METHOD metNotShowChannel : BOOL
VAR_INPUT
    iChannel    :   INT;
END_VAR
IF iChannel >= 1 AND iChannel <= 16 THEN
    metNotShowChannel := NOT ayShowChanel[iChannel];
ELSE
    metNotShowChannel := TRUE;
END_IF
END_METHOD

PROPERTY proScrollBar : INT
SET
iScrollBar := proScrollBar;
END_SET
GET
proScrollBar := iOldScrollBar;
END_GET
END_PROPERTY

METHOD PRIVATE metCalcScrollBar : INT
VAR_INPUT
    usiSlot :   USINT;
END_VAR
IF usiSlot <= 11 THEN
    metCalcScrollBar := 0;
ELSE
    metCalcScrollBar := TO_INT(LIMIT(0,((usiSlot -11)* TO_INT(rFactor * 49)),TO_INT(rFactor *2921)));
END_IF;
END_METHOD

METHOD PRIVATE metCalcSlotFromScrollBar : USINT
VAR_INPUT
    iScrollBarIn  :   INT;
END_VAR
IF iScrollBarIn / 49 <= 11 THEN
    metCalcSlotFromScrollBar := 11;
ELSE
    metCalcSlotFromScrollBar := TO_USINT(iScrollBarIn / MAX(1,TO_INT(rFactor*49)));
END_IF;
END_METHOD

METHOD getSizeOfFrame : BOOL
VAR_INPUT
	ptIn	:	VisuElems.VisuStructPoint;
END_VAR
getSizeOfFrame := FALSE;
iFrameSize := ptIn.iX;

IF iFrameSize > 0 THEN
	rFactor := TO_REAL(iFrameSize) / 3000.0;
ELSE
	rFactor := 0;
END_IF
END_METHOD

END_FUNCTION_BLOCK

// 40 Visualizations/AI/SimAI_Temp
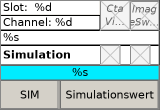
VISUALIZATION SimAI_Temp  // 160x110
VAR_INPUT
	ITF_AI : ITF_AI;
END_VAR
VAR_IN_OUT
	IO_Ref_In	:	fbAI;
END_VAR
    Frame (0,0 160x45)
        shows ModulInfos(ITF_IO := ITF_AI)
    Frame (0,45 160x20)
        shows SimulationInfos(ITF_IO_REF_IN := ITF_AI.proThisRef_AI)
    Textfield (0,65 160x15), "%s", text variable: ITF_AI.proPhysikalValueVisu
    Button (0,80 60x30), "SIM", colour toggle: IO_Ref_In.fbxSimulation.xValue, pressed state: IO_Ref_In.fbxSimulation.xValue, invisible if: IO_Ref_In.fbxSimulationLock.xValue
        toggle IO_Ref_In.fbxSimulation.xValue
    Button (60,80 100x30), "Simulationswert", text variable: IO_Ref_In.fbrSimulationValue.rValue, invisible if: IO_Ref_In.fbxSimulationLock.xValue OR NOT IO_Ref_In.fbxSimulation.xValue
        OnMouseClick: write the text variable via InputWithLimits, min GlobalKonstant.ayMin[ITF_AI.proModuleType], max GlobalKonstant.ayMax[ITF_AI.proModuleType]
END_VISUALIZATION

// 40 Visualizations/AI/SimAI
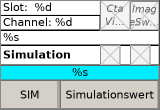
VISUALIZATION SimAI  // 160x110
VAR_INPUT	
	ITF_AI : ITF_AI;
END_VAR
    Frame (0,0 160x110), invisible if: NOT __QUERYINTERFACE(ITF_AI,ITF_AI)
        shows SimAI_Temp_Querry(ITF_AI := ITF_AI)
END_VISUALIZATION

// 40 Visualizations/AO/SimAO_Temp
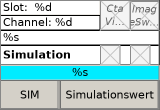
VISUALIZATION SimAO_Temp  // 160x110
VAR_INPUT
	ITF_AO : ITF_AO;
END_VAR
VAR_IN_OUT
	IO_Ref_In	:	fbAO;
END_VAR
    Frame (0,0 160x45)
        shows ModulInfos(ITF_IO := ITF_AO)
    Frame (0,45 160x20)
        shows SimulationInfos(ITF_IO_REF_IN := ITF_AO.proThisRef_AO)
    Textfield (0,65 160x15), "%s", text variable: ITF_AO.proPhysikalValueVisu
    Button (0,80 60x30), "SIM", colour toggle: IO_Ref_In.fbxSimulation.xValue, pressed state: IO_Ref_In.fbxSimulation.xValue, invisible if: IO_Ref_In.fbxSimulationLock.xValue
        toggle IO_Ref_In.fbxSimulation.xValue
    Button (60,80 100x30), "Simulationswert", text variable: IO_Ref_In.fbrSimulationValue.rValue, invisible if: IO_Ref_In.fbxSimulationLock.xValue OR NOT IO_Ref_In.fbxSimulation.xValue
        OnMouseClick: write the text variable via InputWithLimits, min GlobalKonstant.ayMin[ITF_AO.proModuleType], max GlobalKonstant.ayMax[ITF_AO.proModuleType]
END_VISUALIZATION

// 40 Visualizations/AO/SimAO
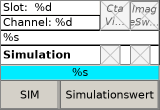
VISUALIZATION SimAO  // 160x110
VAR_INPUT	
	ITF_AO : ITF_AO;
END_VAR
    Frame (0,0 160x110), invisible if: NOT __QUERYINTERFACE(ITF_AO,ITF_AO)
        shows SimAO_Temp_Querry(ITF_AO := ITF_AO)
END_VISUALIZATION

// 40 Visualizations/DI/SimDI
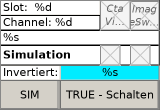
VISUALIZATION SimDI  // 160x110
VAR_INPUT	
	ITF_DI : ITF_DI;
END_VAR
    Frame (0,0 160x110), invisible if: NOT __QUERYINTERFACE(ITF_DI,ITF_DI)
        shows SimDI_Temp_Querry(ITF_DI := ITF_DI)
END_VISUALIZATION

// 40 Visualizations/DI/SimDI_Temp
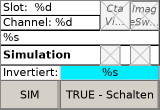
VISUALIZATION SimDI_Temp  // 160x110
VAR_INPUT
	ITF_DI : ITF_DI;
END_VAR
VAR_IN_OUT
	IO_Ref_In	:	fbDI;
END_VAR
    Textfield (0,65 60x15), colour toggle: IO_Ref_In.fbxInvert.xValue
    Textfield (60,65 100x15), "%s", text variable: ITF_DI.proPhysikalValueVisu
    Label (0,65 60x15), "Invertiert:", invisible if: NOT IO_Ref_In.fbxInvert.xValue
    Button (0,80 60x30), "SIM", colour toggle: IO_Ref_In.fbxSimulation.xValue, pressed state: IO_Ref_In.fbxSimulation.xValue, invisible if: IO_Ref_In.fbxSimulationLock.xValue
        toggle IO_Ref_In.fbxSimulation.xValue
    Button (60,80 100x30), "FALSE - Schalten", pressed state: IO_Ref_In.fbxSimulationValue.xValue, invisible if: IO_Ref_In.fbxSimulationLock.xValue OR NOT IO_Ref_In.fbxSimulation.xValue OR NOT IO_Ref_In.fbxSimulationValue.xValue OR IO_Ref_In.fbxInvert.xValue
        toggle IO_Ref_In.fbxSimulationValue.xValue p2164770859=TRUE
    Frame (0,0 160x45)
        shows ModulInfos(ITF_IO := ITF_DI)
    Frame (0,45 160x20)
        shows SimulationInfos(ITF_IO_REF_IN := ITF_DI.proThisRef_DI)
    Button (60,80 100x30), "TRUE - Schalten", pressed state: IO_Ref_In.fbxSimulationValue.xValue, invisible if: IO_Ref_In.fbxSimulationLock.xValue OR NOT IO_Ref_In.fbxSimulation.xValue OR IO_Ref_In.fbxSimulationValue.xValue OR IO_Ref_In.fbxInvert.xValue
        toggle IO_Ref_In.fbxSimulationValue.xValue
    Button (60,80 100x30), "FALSE - Schalten", pressed state: IO_Ref_In.fbxSimulationValue.xValue, invisible if: IO_Ref_In.fbxSimulationLock.xValue OR NOT IO_Ref_In.fbxSimulation.xValue OR IO_Ref_In.fbxSimulationValue.xValue OR NOT IO_Ref_In.fbxInvert.xValue
        toggle IO_Ref_In.fbxSimulationValue.xValue
    Button (60,80 100x30), "TRUE - Schalten", pressed state: IO_Ref_In.fbxSimulationValue.xValue, invisible if: IO_Ref_In.fbxSimulationLock.xValue OR NOT IO_Ref_In.fbxSimulation.xValue OR NOT IO_Ref_In.fbxSimulationValue.xValue OR NOT IO_Ref_In.fbxInvert.xValue
        toggle IO_Ref_In.fbxSimulationValue.xValue
END_VISUALIZATION

// 40 Visualizations/DO/SimDO_Temp
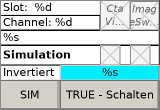
VISUALIZATION SimDO_Temp  // 160x110
VAR_INPUT	
	ITF_DO : ITF_DO;
END_VAR
VAR_IN_OUT
	IO_Ref_In	:	fbDO;
END_VAR
    Textfield (0,65 60x15), colour toggle: IO_Ref_In.fbxInvert.xValue
    Frame (0,0 160x45)
        shows ModulInfos(ITF_IO := ITF_DO)
    Frame (0,45 160x20)
        shows SimulationInfos(ITF_IO_REF_IN := ITF_DO.proThisRef_DO)
    Textfield (60,65 100x15), "%s", text variable: ITF_DO.proPhysikalValueVisu
    Label (0,65 60x15), "Invertiert", invisible if: NOT IO_Ref_In.fbxInvert.xValue
    Button (0,80 60x30), "SIM", colour toggle: IO_Ref_In.fbxSimulation.xValue, pressed state: IO_Ref_In.fbxSimulation.xValue, invisible if: IO_Ref_In.fbxSimulationLock.xValue
        toggle IO_Ref_In.fbxSimulation.xValue
    Button (60,80 100x30), "FALSE - Schalten", pressed state: IO_Ref_In.fbxSimulationValue.xValue, invisible if: IO_Ref_In.fbxSimulationLock.xValue OR NOT IO_Ref_In.fbxSimulation.xValue OR NOT IO_Ref_In.fbxSimulationValue.xValue OR IO_Ref_In.fbxInvert.xValue
        toggle IO_Ref_In.fbxSimulationValue.xValue
    Button (60,80 100x30), "TRUE - Schalten", pressed state: IO_Ref_In.fbxSimulationValue.xValue, invisible if: IO_Ref_In.fbxSimulationLock.xValue OR NOT IO_Ref_In.fbxSimulation.xValue OR IO_Ref_In.fbxSimulationValue.xValue OR IO_Ref_In.fbxInvert.xValue
        toggle IO_Ref_In.fbxSimulationValue.xValue
    Button (60,80 100x30), "FALSE - Schalten", pressed state: IO_Ref_In.fbxSimulationValue.xValue, invisible if: IO_Ref_In.fbxSimulationLock.xValue OR NOT IO_Ref_In.fbxSimulation.xValue OR IO_Ref_In.fbxSimulationValue.xValue OR NOT IO_Ref_In.fbxInvert.xValue
        toggle IO_Ref_In.fbxSimulationValue.xValue
    Button (60,80 100x30), "TRUE - Schalten", pressed state: IO_Ref_In.fbxSimulationValue.xValue, invisible if: IO_Ref_In.fbxSimulationLock.xValue OR NOT IO_Ref_In.fbxSimulation.xValue OR NOT IO_Ref_In.fbxSimulationValue.xValue OR NOT IO_Ref_In.fbxInvert.xValue
        toggle IO_Ref_In.fbxSimulationValue.xValue
END_VISUALIZATION

// 40 Visualizations/DO/SimDO
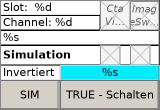
VISUALIZATION SimDO  // 160x110
VAR_INPUT	
	ITF_DO : ITF_DO;
END_VAR
    Frame (0,0 160x110), invisible if: NOT __QUERYINTERFACE(ITF_DO,ITF_DO)
        shows SimDO_Temp_Querry(ITF_DO := ITF_DO)
END_VISUALIZATION

// 40 Visualizations/PFC VISU/IO_ManagerBusInfo
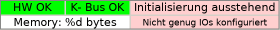
VISUALIZATION IO_ManagerBusInfo  // 280x30
VAR_INPUT
	xErrNotEnoughIOs	:	BOOL;
	xIoInitDone		    : 	BOOL;
	xKbusErrHW		    :	BOOL;
	xKbusErrSW		    : 	BOOL;
	udiNeededMemSize	: 	UDINT;
END_VAR
    Textfield (0,0 65x15), "HW Error", invisible if: NOT xKbusErrHW
    Textfield (0,0 65x15), "HW OK", invisible if: xKbusErrHW
    Textfield (65,0 65x15), "Reboot", invisible if: NOT xKbusErrSW
    Textfield (0,15 130x15), "Memory: %d bytes", text variable: udiNeededMemSize
    Textfield (130,15 150x15), "OK", invisible if: xErrNotEnoughIOs
    Textfield (130,15 150x15), "Nicht genug IOs konfiguriert", invisible if: NOT xErrNotEnoughIOs
    Textfield (130,0 150x15), "Initialisierung erfolgreich", invisible if: NOT xIoInitDone
    Textfield (130,0 150x15), "Initialisierung ausstehend", invisible if: xIoInitDone
    Textfield (65,0 65x15), "K- Bus OK", invisible if: xKbusErrSW
END_VISUALIZATION

// 40 Visualizations/Simulation/Simulation
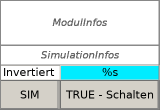
VISUALIZATION Simulation  // 160x110
VAR_INPUT	
	ITF_IO : ITF_IO;
END_VAR

VAR
	ITF_DI 	:	ITF_DI;
	ITF_DO 	:	ITF_DO;
	ITF_AI	:	ITF_AI;
	ITF_AO	:	ITF_AO;
END_VAR
    Frame (0,0 160x110), invisible if: NOT __QUERYINTERFACE(ITF_IO,ITF_DI)
        shows SimDI(ITF_DI := ITF_DI)
    Frame (0,0 160x110), invisible if: NOT __QUERYINTERFACE(ITF_IO,ITF_AI)
        shows SimAI(ITF_AI := ITF_AI)
    Frame (0,0 160x110), invisible if: NOT __QUERYINTERFACE(ITF_IO,ITF_AO)
        shows SimAO(ITF_AO := ITF_AO)
    Frame (0,0 160x110), invisible if: NOT __QUERYINTERFACE(ITF_IO,ITF_DO)
        shows SimDO(ITF_DO := ITF_DO)
END_VISUALIZATION

// 40 Visualizations/Simulation/ModulInfos
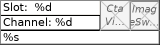
VISUALIZATION ModulInfos  // 160x45
VAR_INPUT	
	ITF_IO : ITF_IO;
END_VAR
    Textfield (0,0 100x15), "Slot: %d", text variable: ITF_IO.proSlot
    Textfield (0,15 100x15), "Channel: %d", text variable: ITF_IO.proChannel
    Textfield (0,30 160x15), "%s", text list: 'txtModulType', text index: ITF_IO.proModuleType
    Rectangle (130,0 30x30)
    ImageSwitcher (130,1 29x29), variable: ITF_IO.proOK, input disabled if: TRUE, background image: CtaVisSymbols.ImagePool.check_green, image: CtaVisSymbols.ImagePool.CtaError, behaviour: TOGGLE
    Rectangle (100,0 30x30)
    Image (100,0 30x30), image: CtaVisSymbols.ImagePool.gear
        OnMouseClick:  Dialog=DIA_IO_CONFIG, Parameters={ITF_IO_IN: ITF_IO}, OpenModal=True, OpenCentered=True
END_VISUALIZATION

// 40 Visualizations/Simulation/SimulationInfos
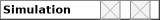
VISUALIZATION SimulationInfos  // 160x20
VAR_IN_OUT
	ITF_IO_REF_IN : fbIO;
END_VAR
    Rectangle (0,0 160x20)
    Label (0,0 100x20), "Simulation", invisible if: ITF_IO_REF_IN.fbxSimulationLock.xValue
    ImageSwitcher (130,0 20x20), variable: ITF_IO_REF_IN.fbxSimulationLock.xValue, input disabled if: TRUE, background image: CtaVisSymbols.ImagePool.lock_closed_black, image: CtaVisSymbols.ImagePool.lock_open_black, behaviour: TOGGLE
    ImageSwitcher (100,0 20x20), variable: ITF_IO_REF_IN.fbxSimulation.xValue, invisible if: ITF_IO_REF_IN.fbxSimulationLock.xValue, input disabled if: TRUE, background image: CtaVisSymbols.ImagePool.front_hand_Yellow, image: CtaVisSymbols.ImagePool.front_hand_Black, behaviour: TOGGLE
END_VISUALIZATION

// 40 Visualizations/Parameter/VIS_IO_PARAMETER_BASE
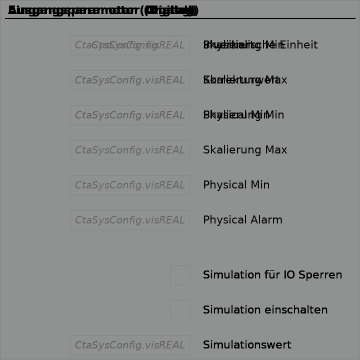
VISUALIZATION VIS_IO_PARAMETER_BASE  // 360x360
VAR_INPUT
    ITF_IO_IN 	: 	ITF_IO;
END_VAR
VAR
	ITF_AI 		:	ITF_AI;
	ITF_DI		:	ITF_DI;
	ITF_AO		:	ITF_AO;
	ITF_DO		:	ITF_DO;
END_VAR
    Frame (0,0 360x360), invisible if: NOT __QUERYINTERFACE(ITF_IO_IN,ITF_AI)
        shows VIS_PARAMETER_AI(ITF_AI_IN := ITF_AI)
        shows VIS_PARAMETER_AO(ITF_AO_IN := ITF_AO)
        shows VIS_PARAMETER_DI(ITF_DI_IN := ITF_DI)
        shows VIS_PARAMETER_DO(ITF_DO_IN := ITF_DO)
        p1531675999: ITF_SENSOR_IN.proThisReference
    Frame (0,0 360x360), invisible if: NOT __QUERYINTERFACE(ITF_IO_IN,ITF_AO)
        shows VIS_PARAMETER_AO(ITF_AO_IN := ITF_AO)
        shows VIS_PARAMETER_AO(ITF_AO_IN := ITF_AO)
        shows VIS_PARAMETER_DI(ITF_DI_IN := ITF_DI)
        shows VIS_PARAMETER_DO(ITF_DO_IN := ITF_DO)
        p1531675999: ITF_SENSOR_IN.proThisReference
    Frame (0,0 360x360), invisible if: NOT __QUERYINTERFACE(ITF_IO_IN,ITF_DI)
        shows VIS_PARAMETER_DI(ITF_DI_IN := ITF_DI)
        shows VIS_PARAMETER_AO(ITF_AO_IN := ITF_AO)
        shows VIS_PARAMETER_DI(ITF_DI_IN := ITF_DI)
        shows VIS_PARAMETER_DO(ITF_DO_IN := ITF_DO)
        p1531675999: ITF_SENSOR_IN.proThisReference
    Frame (0,0 360x360), invisible if: NOT __QUERYINTERFACE(ITF_IO_IN,ITF_DO)
        shows VIS_PARAMETER_DO(ITF_DO_IN := ITF_DO)
        shows VIS_PARAMETER_AO(ITF_AO_IN := ITF_AO)
        shows VIS_PARAMETER_DI(ITF_DI_IN := ITF_DI)
        shows VIS_PARAMETER_DO(ITF_DO_IN := ITF_DO)
        p1531675999: ITF_SENSOR_IN.proThisReference
END_VISUALIZATION

// 40 Visualizations/Parameter/Parameter_AI/VIS_PARAMETER_AI
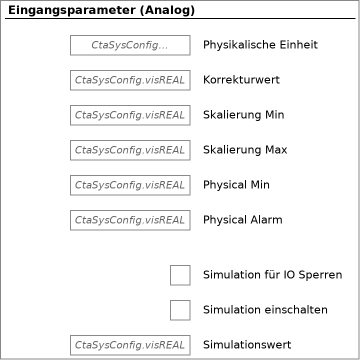
VISUALIZATION VIS_PARAMETER_AI  // 360x360
VAR_INPUT
    ITF_AI_IN	:  	ITF_AI;
END_VAR
    Frame (0,0 360x360), invisible if: NOT __QUERYINTERFACE(ITF_AI_IN,ITF_AI_IN)
        shows VIS_PARAMETER_TEMP_AI(ITF_AI_IN := ITF_AI_IN)
END_VISUALIZATION

// 40 Visualizations/Parameter/Parameter_AI/VIS_PARAMETER_TEMP_AI
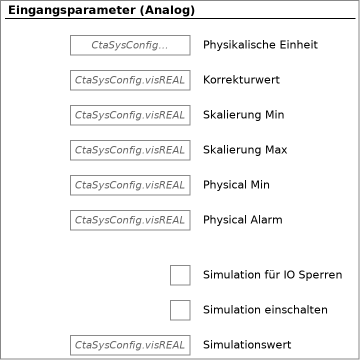
VISUALIZATION VIS_PARAMETER_TEMP_AI  // 360x360
VAR_INPUT
    ITF_AI_IN	:  	ITF_AI;
END_VAR
    Label (5,0 350x20), "Eingangsparameter (Analog)"
    Line (5,18) (355,18)
    Frame (70,35 120x20), invisible if: ITF_AI_IN.proModuleType = 7
        shows CtaSysConfig.visSTRING40(visfbSTRING40In := ITF_AI_IN.P_scfbAI_fbstPhysicalUnit)
    Label (200,35 150x20), "Physikalische Einheit", invisible if: ITF_AI_IN.proModuleType = 7
    Frame (70,70 120x20)
        shows CtaSysConfig.visREAL(visfbREALIn := ITF_AI_IN.P_scfbAI_fbrCorrectionValue, stPhysikalischeEinheit := CtaSysConfig.fcGetValueFromDataType(ITF_AI_IN.P_scfbAI_fbstPhysicalUnit))
    Label (200,70 150x20), "Korrekturwert"
    Frame (70,105 120x20), invisible if: ITF_AI_IN.proModuleType = 7
        shows CtaSysConfig.visREAL(visfbREALIn := ITF_AI_IN.P_scfbAI_fbrMin, stPhysikalischeEinheit := CtaSysConfig.fcGetValueFromDataType(ITF_AI_IN.P_scfbAI_fbstPhysicalUnit))
    Label (200,105 150x20), "Skalierung Min", invisible if: ITF_AI_IN.proModuleType = 7
    Frame (70,140 120x20), invisible if: ITF_AI_IN.proModuleType = 7
        shows CtaSysConfig.visREAL(visfbREALIn := ITF_AI_IN.P_scfbAI_fbrMax, stPhysikalischeEinheit := CtaSysConfig.fcGetValueFromDataType(ITF_AI_IN.P_scfbAI_fbstPhysicalUnit))
    Label (200,140 150x20), "Skalierung Max", invisible if: ITF_AI_IN.proModuleType = 7
    Frame (70,175 120x20), invisible if: ITF_AI_IN.proModuleType <> 5
        shows CtaSysConfig.visREAL(visfbREALIn := ITF_AI_IN.P_scfbAI_fbrMinPhysical, stPhysikalischeEinheit := 'V')
    Label (200,175 150x20), "Physical Min", invisible if: ITF_AI_IN.proModuleType <> 5
    Frame (70,210 120x20), invisible if: ITF_AI_IN.proModuleType <> 5
        shows CtaSysConfig.visREAL(visfbREALIn := ITF_AI_IN.P_scfbAI_fbrPhysicalAlarm, stPhysikalischeEinheit := 'V')
    Label (200,210 150x20), "Physical Alarm", invisible if: ITF_AI_IN.proModuleType <> 5
    Frame (70,335 120x20), invisible if: CtaSysConfig.fcGetEnumerationId(ITF_AI_IN.P_scfbIO_fbxSimulationLock) = 1
        shows CtaSysConfig.visREAL(visfbREALIn := ITF_AI_IN.P_scfbAI_fbrSimulationValue)
    Label (200,335 150x20), "Simulationswert", invisible if: CtaSysConfig.fcGetEnumerationId(ITF_AI_IN.P_scfbIO_fbxSimulationLock) = 1
    Label (200,300 150x20), "Simulation einschalten", invisible if: CtaSysConfig.fcGetEnumerationId(ITF_AI_IN.P_scfbIO_fbxSimulationLock) = 1
    Label (200,265 150x20), "Simulation für IO Sperren"
    Frame (170,265 20x20)
        shows CtaSysConfig.visBOOL(visfbBOOLIn := ITF_AI_IN.P_scfbIO_fbxSimulationLock)
    Frame (170,300 20x20), invisible if: CtaSysConfig.fcGetEnumerationId(ITF_AI_IN.P_scfbIO_fbxSimulationLock) = 1
        shows CtaSysConfig.visBOOL(visfbBOOLIn := ITF_AI_IN.P_scfbIO_Simulation)
    Textfield (295,335 60x20), text list: 'txtPhysicalUnit', text index: TO_STRING(TO_INT(ITF_AI_IN.proModuleType))
END_VISUALIZATION

// 40 Visualizations/Parameter/Parameter_DI/VIS_PARAMETER_DI
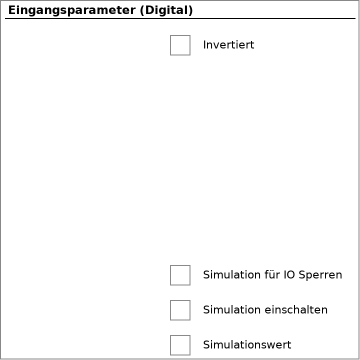
VISUALIZATION VIS_PARAMETER_DI  // 360x360
VAR_INPUT
    ITF_DI_IN	:  	ITF_DI;
END_VAR
    Frame (0,0 360x360), invisible if: NOT __QUERYINTERFACE(ITF_DI_IN,ITF_DI_IN)
        shows VIS_PARAMETER_TEMP_DI(ITF_DI_IN := ITF_DI_IN)
        pReferences[0]: IO_REF_IN=ITF_AI_IN.proThisRef_AI
END_VISUALIZATION

// 40 Visualizations/Parameter/Parameter_DI/VIS_PARAMETER_TEMP_DI
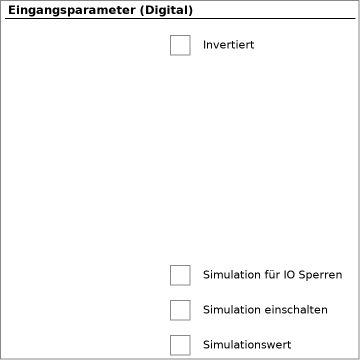
VISUALIZATION VIS_PARAMETER_TEMP_DI  // 360x360
VAR_INPUT
    ITF_DI_IN	:  	ITF_DI;
END_VAR
    Label (5,0 350x20), "Eingangsparameter (Digital)"
    Line (5,18) (355,18)
    Frame (170,35 20x20)
        shows CtaSysConfig.visBOOL(visfbBOOLIn := ITF_DI_IN.P_scfbDI_fbxInvert)
    Label (200,35 150x20), "Invertiert"
    Frame (170,335 20x20), invisible if: CtaSysConfig.fcGetEnumerationId(ITF_DI_IN.P_scfbIO_fbxSimulationLock) = 1
        shows CtaSysConfig.visBOOL(visfbBOOLIn := ITF_DI_IN.P_scfbDI_fbxSimulationValue)
    Label (200,335 150x20), "Simulationswert", invisible if: CtaSysConfig.fcGetEnumerationId(ITF_DI_IN.P_scfbIO_fbxSimulationLock) = 1
    Frame (170,265 20x20)
        shows CtaSysConfig.visBOOL(visfbBOOLIn := ITF_DI_IN.P_scfbIO_fbxSimulationLock)
    Label (200,300 150x20), "Simulation einschalten", invisible if: CtaSysConfig.fcGetEnumerationId(ITF_DI_IN.P_scfbIO_fbxSimulationLock) = 1
    Label (200,265 150x20), "Simulation für IO Sperren"
    Frame (170,300 20x20), invisible if: CtaSysConfig.fcGetEnumerationId(ITF_DI_IN.P_scfbIO_fbxSimulationLock) = 1
        shows CtaSysConfig.visBOOL(visfbBOOLIn := ITF_DI_IN.P_scfbIO_Simulation)
END_VISUALIZATION

// 40 Visualizations/AI/SimAI_Temp_Querry
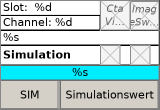
VISUALIZATION SimAI_Temp_Querry  // 160x110
VAR_INPUT
	ITF_AI : ITF_AI;
END_VAR
    Frame (0,0 160x110)
        shows SimAI_Temp(ITF_AI := ITF_AI, IO_Ref_In := ITF_AI.proThisRef_AI)
END_VISUALIZATION

// 40 Visualizations/AO/SimAO_Temp_Querry
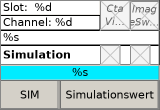
VISUALIZATION SimAO_Temp_Querry  // 160x110
VAR_INPUT
	ITF_AO : ITF_AO;
END_VAR
    Frame (0,0 160x110)
        shows SimAO_Temp(ITF_AO := ITF_AO, IO_Ref_In := ITF_AO.proThisRef_AO)
END_VISUALIZATION

// 40 Visualizations/Parameter/Parameter_AO/VIS_PARAMETER_AO
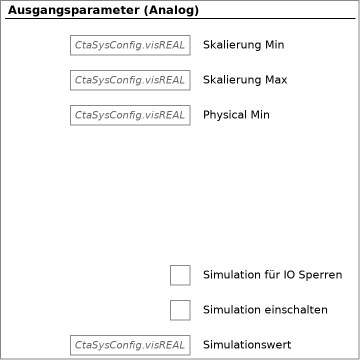
VISUALIZATION VIS_PARAMETER_AO  // 360x360
VAR_INPUT
    ITF_AO_IN	:  	ITF_AO;
END_VAR
    Frame (0,0 360x360), invisible if: NOT __QUERYINTERFACE(ITF_AO_IN,ITF_AO_IN)
        shows VIS_PARAMETER_TEMP_AO(ITF_AO_IN := ITF_AO_IN)
END_VISUALIZATION

// 40 Visualizations/Parameter/Parameter_AO/VIS_PARAMETER_TEMP_AO
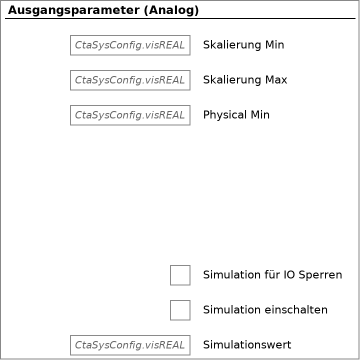
VISUALIZATION VIS_PARAMETER_TEMP_AO  // 360x360
VAR_INPUT
    ITF_AO_IN	:  	ITF_AO;
END_VAR
    Label (5,0 350x20), "Ausgangsparameter (Analog)"
    Line (5,18) (355,18)
    Frame (70,35 120x20)
        shows CtaSysConfig.visREAL(visfbREALIn := ITF_AO_IN.P_scfbAO_fbrMin)
    Label (200,35 150x20), "Skalierung Min"
    Frame (70,70 120x20)
        shows CtaSysConfig.visREAL(visfbREALIn := ITF_AO_IN.P_scfbAO_fbrMax)
    Label (200,70 150x20), "Skalierung Max"
    Frame (70,105 120x20)
        shows CtaSysConfig.visREAL(visfbREALIn := ITF_AO_IN.P_scfbAO_fbrMinPhysical)
    Label (200,105 150x20), "Physical Min"
    Frame (70,335 120x20), invisible if: CtaSysConfig.fcGetEnumerationId(ITF_AO_IN.P_scfbIO_fbxSimulationLock) = 1
        shows CtaSysConfig.visREAL(visfbREALIn := ITF_AO_IN.P_scfbAO_fbrSimulationValue)
    Label (200,335 150x20), "Simulationswert", invisible if: CtaSysConfig.fcGetEnumerationId(ITF_AO_IN.P_scfbIO_fbxSimulationLock) = 1
    Frame (170,265 20x20)
        shows CtaSysConfig.visBOOL(visfbBOOLIn := ITF_AO_IN.P_scfbIO_fbxSimulationLock)
    Label (200,300 150x20), "Simulation einschalten", invisible if: CtaSysConfig.fcGetEnumerationId(ITF_AO_IN.P_scfbIO_fbxSimulationLock) = 1
    Label (200,265 150x20), "Simulation für IO Sperren"
    Frame (170,300 20x20), invisible if: CtaSysConfig.fcGetEnumerationId(ITF_AO_IN.P_scfbIO_fbxSimulationLock) = 1
        shows CtaSysConfig.visBOOL(visfbBOOLIn := ITF_AO_IN.P_scfbIO_Simulation)
    Textfield (295,335 60x20), text list: 'txtPhysicalUnit', text index: TO_STRING(TO_INT(ITF_AO_IN.proModuleType))
END_VISUALIZATION

// 40 Visualizations/Parameter/Parameter_DO/VIS_PARAMETER_DO
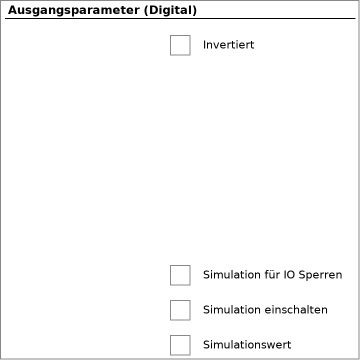
VISUALIZATION VIS_PARAMETER_DO  // 360x360
VAR_INPUT
    ITF_DO_IN	:  	ITF_DO;
END_VAR
    Frame (0,0 360x360), invisible if: NOT __QUERYINTERFACE(ITF_DO_IN,ITF_DO_IN)
        shows VIS_PARAMETER_TEMP_DO(ITF_DO_IN := ITF_DO_IN)
END_VISUALIZATION

// 40 Visualizations/Parameter/Parameter_DO/VIS_PARAMETER_TEMP_DO
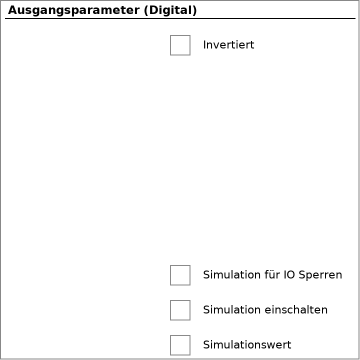
VISUALIZATION VIS_PARAMETER_TEMP_DO  // 360x360
VAR_INPUT
    ITF_DO_IN	:  	ITF_DO;
END_VAR
    Label (5,0 350x20), "Ausgangsparameter (Digital)"
    Line (5,18) (355,18)
    Frame (170,35 20x20)
        shows CtaSysConfig.visBOOL(visfbBOOLIn := ITF_DO_IN.P_scfbDO_fbxInvert)
    Label (200,35 150x20), "Invertiert"
    Frame (170,335 20x20), invisible if: CtaSysConfig.fcGetEnumerationId(ITF_DO_IN.P_scfbIO_fbxSimulationLock) = 1
        shows CtaSysConfig.visBOOL(visfbBOOLIn := ITF_DO_IN.P_scfbDO_fbxSimulationValue)
    Label (200,335 150x20), "Simulationswert", invisible if: CtaSysConfig.fcGetEnumerationId(ITF_DO_IN.P_scfbIO_fbxSimulationLock) = 1
    Frame (170,265 20x20)
        shows CtaSysConfig.visBOOL(visfbBOOLIn := ITF_DO_IN.P_scfbIO_fbxSimulationLock)
    Label (200,300 150x20), "Simulation einschalten", invisible if: CtaSysConfig.fcGetEnumerationId(ITF_DO_IN.P_scfbIO_fbxSimulationLock) = 1
    Label (200,265 150x20), "Simulation für IO Sperren"
    Frame (170,300 20x20), invisible if: CtaSysConfig.fcGetEnumerationId(ITF_DO_IN.P_scfbIO_fbxSimulationLock) = 1
        shows CtaSysConfig.visBOOL(visfbBOOLIn := ITF_DO_IN.P_scfbIO_Simulation)
END_VISUALIZATION

// 40 Visualizations/DI/SimDI_Temp_Querry
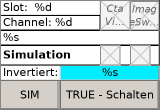
VISUALIZATION SimDI_Temp_Querry  // 160x110
VAR_INPUT
	ITF_DI : ITF_DI;
END_VAR
    Frame (0,0 160x110)
        shows SimDI_Temp(ITF_DI := ITF_DI, IO_Ref_In := ITF_DI.proThisRef_DI)
END_VISUALIZATION

// 40 Visualizations/DO/SimDO_Temp_Querry
